{attribute 'GeneratedUsingTerminal: EL6224-0000-0016'}
{attribute addProperty BoxType "EL6224-0000-0016"}
{attribute addProperty Id "DeviceState_InputsAT %I*DeviceState_Inputs_4751FF764IO_Inputs_Channel_1EMPTY_STRUCTURE0IO_Inputs_Channel_2EMPTY_STRUCTURE0IO_Inputs_Channel_3EMPTY_STRUCTURE0IO_Inputs_Channel_4EMPTY_STRUCTURE0IO_Outputs_Channel_1EMPTY_STRUCTURE0IO_Outputs_Channel_2EMPTY_STRUCTURE0IO_Outputs_Channel_3EMPTY_STRUCTURE0IO_Outputs_Channel_4EMPTY_STRUCTURE0WcStateAT %I*WcState_9091E0EB2InfoDataAT %I*InfoData_90184F0C16"}
{attribute addProperty CRC "3757815554"}
{attribute addProperty Size "22"}
TYPE EL6224_DFFBB702 EXTENDS EtcSlaveTerminalBase_947E5A46 :
STRUCT
	{attribute addProperty Name "DeviceState_Inputs"}
	DeviceState_Inputs : DeviceState_Inputs_4751FF76;
	{attribute addProperty Name "IO_Inputs_Channel_1"}
	IO_Inputs_Channel_1 : EMPTY_STRUCTURE;
	{attribute addProperty Name "IO_Inputs_Channel_2"}
	IO_Inputs_Channel_2 : EMPTY_STRUCTURE;
	{attribute addProperty Name "IO_Inputs_Channel_3"}
	IO_Inputs_Channel_3 : EMPTY_STRUCTURE;
	{attribute addProperty Name "IO_Inputs_Channel_4"}
	IO_Inputs_Channel_4 : EMPTY_STRUCTURE;
	{attribute addProperty Name "IO_Outputs_Channel_1"}
	IO_Outputs_Channel_1 : EMPTY_STRUCTURE;
	{attribute addProperty Name "IO_Outputs_Channel_2"}
	IO_Outputs_Channel_2 : EMPTY_STRUCTURE;
	{attribute addProperty Name "IO_Outputs_Channel_3"}
	IO_Outputs_Channel_3 : EMPTY_STRUCTURE;
	{attribute addProperty Name "IO_Outputs_Channel_4"}
	IO_Outputs_Channel_4 : EMPTY_STRUCTURE;
	{attribute addProperty Name "WcState"}
	WcState : WcState_9091E0EB;
	{attribute addProperty Name "InfoData"}
	InfoData : InfoData_90184F0C;
END_STRUCT
END_TYPE

(* stored: Version 1.2.0.0, ProductVersion 3.1.4024.9
   DUT EL6224_DFFBB702: Id {9646e34f-7066-4b0b-834b-ef02fc33fb85} *)
